FUNCTION_BLOCK FB_CoilCtrl
VAR_INPUT
	i_Interlocks		:ARRAY[1..8] OF BOOL;
	i_ProcesslocksOK	:BOOL;
	i_AutoCmd			:BOOL;
	i_ManCmd			:BOOL;
	i_ServiceMode		:BOOL;
	i_MaintLimit		:UDINT;
	i_PresetValue		:UDINT;
	i_WritePreset		:BOOL;
END_VAR
VAR_OUTPUT
	q_InterlocksOK		:BOOL;
	q_Enabled			:BOOL;
	q_Cmd				:BOOL;
	q_TotalCycles		:UDINT;
	q_MaintCycles		:UDINT;
	q_MaintenanceCall	:BOOL;
END_VAR
VAR
	tofDelayOut			:TOF;
	bCmd				:BOOL;
END_VAR
VAR // added by the converter: edge detectors and wires of the graphical bodies
    _rt1, _rt2 : R_TRIG;
    _w1 : BOOL;
END_VAR

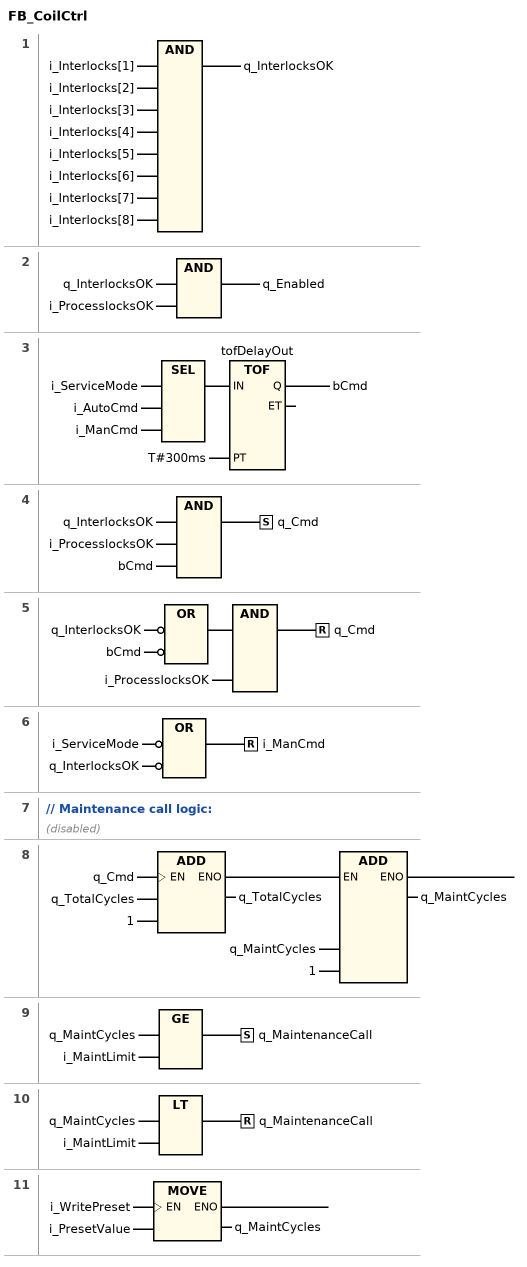
// NETWORK 1
q_InterlocksOK := i_Interlocks[1] AND i_Interlocks[2] AND i_Interlocks[3] AND i_Interlocks[4] AND i_Interlocks[5] AND i_Interlocks[6] AND i_Interlocks[7] AND i_Interlocks[8];

// NETWORK 2
q_Enabled := q_InterlocksOK AND i_ProcesslocksOK;

// NETWORK 3
tofDelayOut(IN := SEL(i_ServiceMode, i_AutoCmd, i_ManCmd), PT := T#300ms); // TOF
bCmd := tofDelayOut.Q;

// NETWORK 4
q_Cmd S= q_InterlocksOK AND i_ProcesslocksOK AND bCmd;

// NETWORK 5
q_Cmd R= (NOT q_InterlocksOK OR NOT bCmd) AND i_ProcesslocksOK;

// NETWORK 6
i_ManCmd R= NOT i_ServiceMode OR NOT q_InterlocksOK;

// NETWORK 7 (disabled)
// label: // Maintenance call logic

// NETWORK 8
_rt1(CLK := q_Cmd);
_w1 := _rt1.Q;
IF _w1 THEN q_TotalCycles := q_TotalCycles + 1; END_IF
IF _w1 THEN q_MaintCycles := q_MaintCycles + 1; END_IF

// NETWORK 9
q_MaintenanceCall S= q_MaintCycles >= i_MaintLimit;

// NETWORK 10
q_MaintenanceCall R= q_MaintCycles < i_MaintLimit;

// NETWORK 11
_rt2(CLK := i_WritePreset);
IF _rt2.Q THEN q_MaintCycles := i_PresetValue; END_IF

END_FUNCTION_BLOCK

(* stored: Version 1.1.0.1, ProductVersion 3.1.4024.12
   POU FB_CoilCtrl: Id {26457a54-c239-458d-bce3-5a4c91c93d54}, SpecialFunc None *)
